// TIA Portal V19 export
TYPE "dtAutoReset"
   STRUCT
      maxAlarms : Int;
      perT : Time;
      autoresetT : Time;
   END_STRUCT;
END_TYPE
